PROGRAM Alarming
VAR
	bInit		: BOOL := TRUE;
	bSendMsg	: BOOL;
	fbMsg		: FB_TcMessage;
END_VAR

IF bInit THEN
	binit := FALSE;
	fbMsg.CreateEx(TC_Events.MyEvents.MyFirstMsg, 0);
END_IF

IF bSendMsg THEN
	bSendMsg := FALSE;
	fbMsg.Send(0);
END_IF

END_PROGRAM

(* stored: Version 1.1.0.1, ProductVersion 3.1.4024.12
   POU Alarming: Id {889a3b90-2598-44bc-a096-5df299aeec61}, SpecialFunc None *)
